KUKA KRL data list: TTT_X.dat

&ACCESS RVO1
&COMMENT
DEFDAT TTT_X PUBLIC
;FOLD EXTERNAL DECLARATIONS;%{PE}%MKUKATPBASIS,%CEXT,%VCOMMON,%P
;FOLD BASISTECH EXT;%{PE}%MKUKATPBASIS,%CEXT,%VEXT,%P
EXT  BAS (BAS_COMMAND  :IN,REAL  :IN )
DECL INT SUCCESS
;ENDFOLD (BASISTECH EXT)
;FOLD USER EXT;%{E}%MKUKATPUSER,%CEXT,%VEXT,%P
;Make here your modifications

;ENDFOLD (USER EXT)
;ENDFOLD (EXTERNAL DECLERATIONS)

DECL INT DELTAX=0
DECL INT DELTAY=0

DECL BASIS_SUGG_T LAST_BASIS={POINT1[] "PTRU",POINT2[] "PTRU",CP_PARAMS[] "CPDAT16",PTP_PARAMS[] "PDAT12",CONT[] " ",CP_VEL[] "1",PTP_VEL[] "100",SYNC_PARAMS[] "SYNCDAT ",SPL_NAME[] "S0 "}
DECL E6POS XPBR={X 100+DELTAX,Y 100+DELTAY,Z 0,A 0,B 0,C 0,S 0,T 0,E1 0,E2 0,E3 0,E4 0,E5 0,E6 0}
DECL FDAT FPBR={TOOL_NO 15,BASE_NO 15,IPO_FRAME #BASE,POINT2[] " ",TQ_STATE FALSE}
DECL LDAT LCPDAT13={VEL 1,ACC 100,APO_DIST 100,APO_FAC 50,AXIS_VEL 100.0,AXIS_ACC 100.0,ORI_TYP #VAR,CIRC_TYP #BASE,JERK_FAC 50.0,GEAR_JERK 50.0,EXAX_IGN 0}
DECL E6POS XPTL={X 0+DELTAX,Y 0+DELTAY,Z 0,A 0,B 0,C 0,S 0,T 0,E1 0,E2 0,E3 0,E4 0,E5 0,E6 0}
DECL FDAT FPTL={TOOL_NO 15,BASE_NO 15,IPO_FRAME #BASE,POINT2[] " ",TQ_STATE FALSE}
DECL LDAT LCPDAT14={VEL 1,ACC 100,APO_DIST 100,APO_FAC 50,AXIS_VEL 100.0,AXIS_ACC 100.0,ORI_TYP #VAR,CIRC_TYP #BASE,JERK_FAC 50.0,GEAR_JERK 50.0,EXAX_IGN 0}
DECL PDAT PPDAT8={VEL 100,ACC 100,APO_DIST 100,APO_MODE #CPTP,GEAR_JERK 50}
DECL E6POS XPBRU={X 100+DELTAX,Y 100+DELTAY,Z -10,A 0,B 0,C 0,S 0,T 0,E1 0,E2 0,E3 0,E4 0,E5 0,E6 0}
DECL FDAT FPBRU={TOOL_NO 15,BASE_NO 15,IPO_FRAME #BASE,POINT2[] " ",TQ_STATE FALSE}
DECL PDAT PPDAT9={VEL 100,ACC 100,APO_DIST 100,APO_MODE #CPTP,GEAR_JERK 50}
DECL E6POS XPBLU={X 0+DELTAX,Y 100+DELTAY,Z -10,A 0,B 0,C 0,S 0,T 0,E1 0,E2 0,E3 0,E4 0,E5 0,E6 0}
DECL FDAT FPBLU={TOOL_NO 15,BASE_NO 15,IPO_FRAME #BASE,POINT2[] " ",TQ_STATE FALSE}
DECL PDAT PPDAT10={VEL 100,ACC 100,APO_DIST 100,APO_MODE #CPTP,GEAR_JERK 50}
DECL E6POS XPBL={X 0+DELTAX,Y 100+DELTAY,Z 0,A 0,B 0,C 0,S 0,T 0,E1 0,E2 0,E3 0,E4 0,E5 0,E6 0}
DECL FDAT FPBL={TOOL_NO 15,BASE_NO 15,IPO_FRAME #BASE,POINT2[] " ",TQ_STATE FALSE}
DECL PDAT PPDAT11={VEL 100,ACC 100,APO_DIST 100,APO_MODE #CPTP,GEAR_JERK 50}
DECL E6POS XPTR={X 100+DELTAX,Y 0+DELTAY,Z 0,A 0,B 0,C 0,S 0,T 0,E1 0,E2 0,E3 0,E4 0,E5 0,E6 0}
DECL FDAT FPTR={TOOL_NO 15,BASE_NO 15,IPO_FRAME #BASE,POINT2[] " ",TQ_STATE FALSE}
DECL LDAT LCPDAT15={VEL 1,ACC 100,APO_DIST 100,APO_FAC 50,AXIS_VEL 100.0,AXIS_ACC 100.0,ORI_TYP #VAR,CIRC_TYP #BASE,JERK_FAC 50.0,GEAR_JERK 50.0,EXAX_IGN 0}
DECL E6POS XPTRU={X 100+DELTAX,Y 0+DELTAY,Z -10,A 0,B 0,C 0,S 0,T 0,E1 0,E2 0,E3 0,E4 0,E5 0,E6 0}
DECL FDAT FPTRU={TOOL_NO 15,BASE_NO 15,IPO_FRAME #BASE,POINT2[] " ",TQ_STATE FALSE}
DECL PDAT PPDAT12={VEL 100,ACC 100,APO_DIST 100,APO_MODE #CPTP,GEAR_JERK 50}
DECL LDAT LCPDAT16={VEL 1,ACC 100,APO_DIST 100,APO_FAC 50,AXIS_VEL 100.0,AXIS_ACC 100.0,ORI_TYP #VAR,CIRC_TYP #BASE,JERK_FAC 50.0,GEAR_JERK 50.0,EXAX_IGN 0}
ENDDAT
